PROGRAM TrendSample
VAR
	VariableForTrend: REAL;
	t: REAL;
	Var1: FB_TrandChanel := (MaximalValue := 1, pPoints := 100);
END_VAR

t:=t+0.01;
VariableForTrend:=SIN(t);
Var1(TrendChannel:= VariableForTrend );

END_PROGRAM

(* stored: Version 1.1.0.1, ProductVersion 3.1.4024.2
   POU TrendSample: Id {cdd5624a-200a-452d-85d1-79574d4adaf6}, SpecialFunc None *)
